FUNCTION_BLOCK T_CheckFileExists
VAR
	fileOpen : FB_FileOpen;
	fileClose : FB_FileClose;
	
	start : BOOL;
	_fileExists : BOOL; 
	
	state : (
		WaitForStart,
		WaitForOpenResult,
		CloseIfOpened
	);
	
END_VAR

CASE state OF
	
	WaitForStart : 
	
		IF start THEN
			 _fileExists := FALSE;
			 state := WaitForOpenResult;
			 start := FALSE;
		END_IF
		
	WaitForOpenResult : 
	
		IF NOT fileOpen.bBusy THEN
			state := SEL( fileOpen.bError, CloseIfOpened, WaitForStart );		
		END_IF
		
	CloseIfOpened : 
	
		IF NOT fileClose.bBusy THEN
			state := WaitForStart;		
		END_IF
		
END_CASE

fileOpen(
	sNetId 		:= '', 
	nMode 		:= FOPEN_MODEREAD,
	bExecute 	:= state = WaitForOpenResult
);
	
fileClose( 
	sNetId := '', 
   hFile := fileOpen.hFile,
	bExecute := state = CloseIfOpened
);
	
_fileExists S= state = CloseIfOpened;

{attribute 'monitoring' := 'variable'}
PROPERTY Busy : BOOL
GET
Busy := 
	start OR ( state <> WaitForStart );
END_GET
END_PROPERTY

METHOD Check
VAR_INPUT
	Path : STRING; // path for new file. 
END_VAR
FileOpen( 
	sPathName := Path
);

start := TRUE;
END_METHOD

{attribute 'monitoring' := 'variable'}
PROPERTY FileExists : BOOL
GET
FileExists := _fileExists AND NOT Busy;
END_GET
END_PROPERTY

END_FUNCTION_BLOCK

(* stored: Version 1.1.0.1, ProductVersion 3.1.4022.18
   POU T_CheckFileExists: Id {10b8c3da-74cc-0d0a-376a-46a39a0c040b}, SpecialFunc None
   Property Busy: Id {a8a19ef0-9ce0-0e75-278d-c2d863ebd11f}
   Get Get: Id {931f9a3e-5ce6-0e39-212c-6c35eb7e3984}
   Method Check: Id {81375c22-709d-0bef-2791-92804698eb08}
   Property FileExists: Id {1ff0828a-3883-01c1-2f1e-f927036791eb}
   Get Get: Id {811ed2f4-b572-04df-236b-344370f21b36} *)
